TYPE FileName : STRING(255);
END_TYPE

(* stored: Version 1.1.0.1, ProductVersion 3.1.4024.9
   DUT FileName: Id {348424eb-a377-41ad-8f1c-40a06d03c436} *)
